PROGRAM MAIN
VAR
END_VAR

PRG_TXI_VAC_GAUGES();
PRG_TXI_VAC_PUMPS();

END_PROGRAM

(* stored: Version 1.1.0.1, ProductVersion 3.1.4024.6
   POU MAIN: Id {aaba3096-245a-4ba7-8aa0-ff7e8fb88c30}, SpecialFunc None *)
